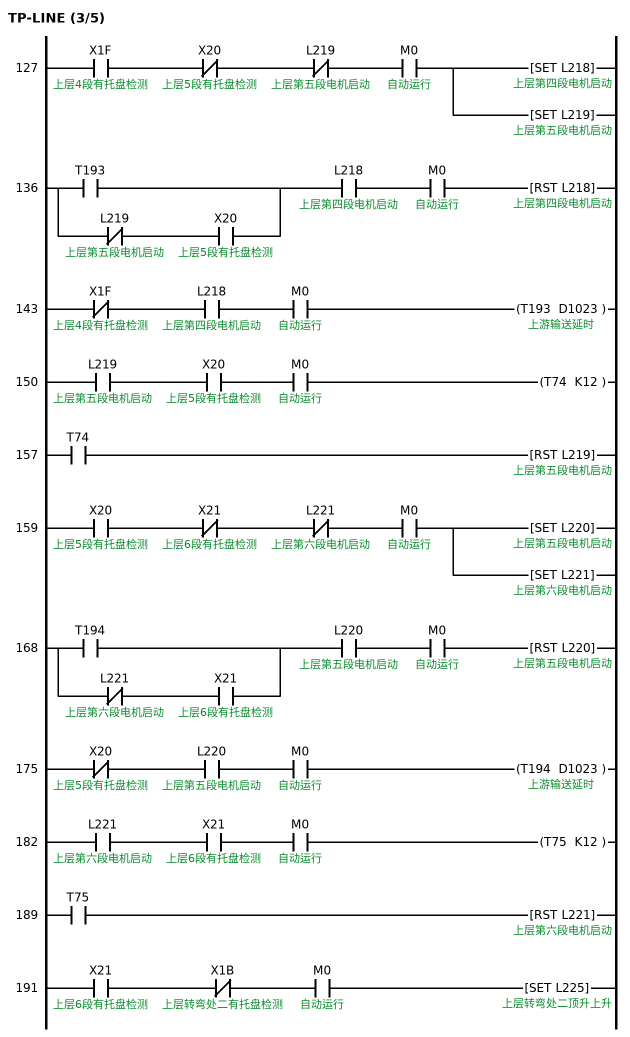
[picture p72: ladder of TP-LINE, rungs at steps 127 to 191]
127   LD      X1F  ; 上层4段有托盘检测
      ANI     X20  ; 上层5段有托盘检测
      ANI     L219  ; 上层第五段电机启动
      AND     M0  ; 自动运行
      SET     L218  ; 上层第四段电机启动
        [note] 5
      SET     L219  ; 上层第五段电机启动
136   LD      T193
      LDI     L219  ; 上层第五段电机启动
      AND     X20  ; 上层5段有托盘检测
      ORB
      AND     L218  ; 上层第四段电机启动
      AND     M0  ; 自动运行
      RST     L218  ; 上层第四段电机启动
143   LDI     X1F  ; 上层4段有托盘检测
      AND     L218  ; 上层第四段电机启动
      AND     M0  ; 自动运行
      OUT     T193 D1023  ; 上游输送延时
150   LD      L219  ; 上层第五段电机启动
      AND     X20  ; 上层5段有托盘检测
      AND     M0  ; 自动运行
      OUT     T74 K12
157   LD      T74
      RST     L219  ; 上层第五段电机启动
159   LD      X20  ; 上层5段有托盘检测
      ANI     X21  ; 上层6段有托盘检测
      ANI     L221  ; 上层第六段电机启动
      AND     M0  ; 自动运行
      SET     L220  ; 上层第五段电机启动
        [note] 6
      SET     L221  ; 上层第六段电机启动
168   LD      T194
      LDI     L221  ; 上层第六段电机启动
      AND     X21  ; 上层6段有托盘检测
      ORB
      AND     L220  ; 上层第五段电机启动
      AND     M0  ; 自动运行
      RST     L220  ; 上层第五段电机启动
175   LDI     X20  ; 上层5段有托盘检测
      AND     L220  ; 上层第五段电机启动
      AND     M0  ; 自动运行
      OUT     T194 D1023  ; 上游输送延时
182   LD      L221  ; 上层第六段电机启动
      AND     X21  ; 上层6段有托盘检测
      AND     M0  ; 自动运行
      OUT     T75 K12
189   LD      T75
      RST     L221  ; 上层第六段电机启动
191   LD      X21  ; 上层6段有托盘检测
      ANI     X1B  ; 上层转弯处二有托盘检测
      AND     M0  ; 自动运行
      SET     L225  ; 上层转弯处二顶升上升
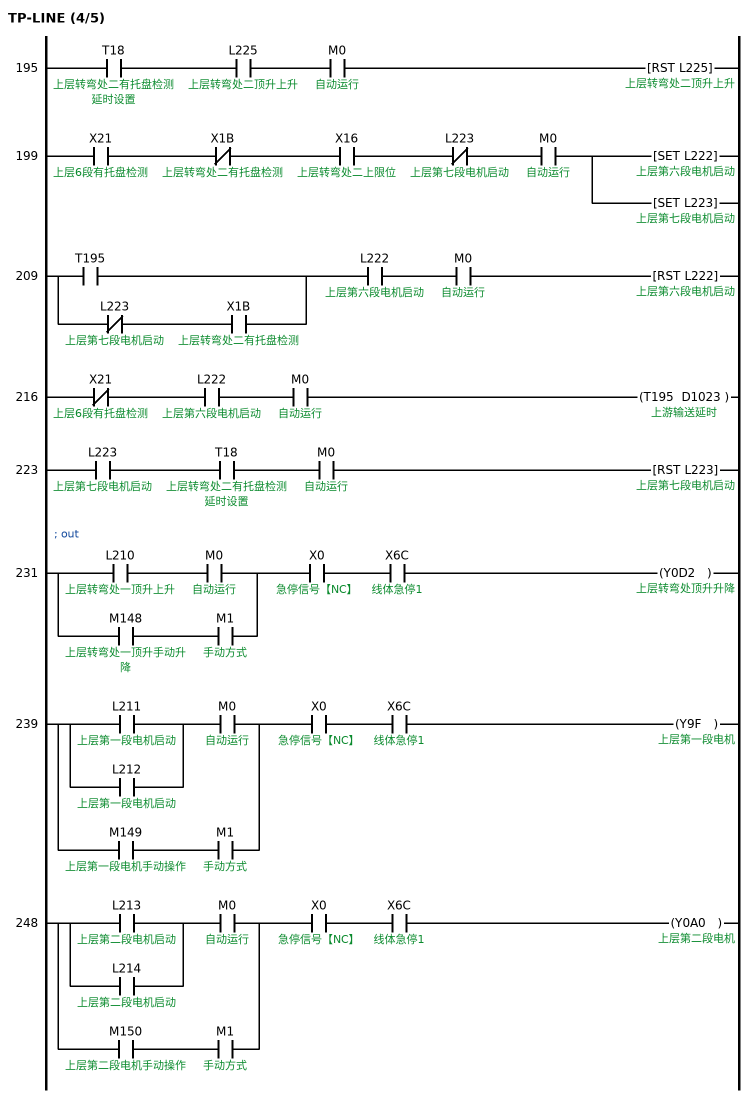
195   LD      T18  ; 上层转弯处二有托盘检测延时设置
      AND     L225  ; 上层转弯处二顶升上升
      AND     M0  ; 自动运行
      RST     L225  ; 上层转弯处二顶升上升
199   LD      X21  ; 上层6段有托盘检测
      ANI     X1B  ; 上层转弯处二有托盘检测
      AND     X16  ; 上层转弯处二上限位
      ANI     L223  ; 上层第七段电机启动
      AND     M0  ; 自动运行
      SET     L222  ; 上层第六段电机启动
        [note] 7
      SET     L223  ; 上层第七段电机启动
209   LD      T195
      LDI     L223  ; 上层第七段电机启动
      AND     X1B  ; 上层转弯处二有托盘检测
      ORB
      AND     L222  ; 上层第六段电机启动
      AND     M0  ; 自动运行
      RST     L222  ; 上层第六段电机启动
216   LDI     X21  ; 上层6段有托盘检测
      AND     L222  ; 上层第六段电机启动
      AND     M0  ; 自动运行
      OUT     T195 D1023  ; 上游输送延时
223   LD      L223  ; 上层第七段电机启动
      AND     T18  ; 上层转弯处二有托盘检测延时设置
      AND     M0  ; 自动运行
      RST     L223  ; 上层第七段电机启动
; out
231   LD      L210  ; 上层转弯处一顶升上升
      AND     M0  ; 自动运行
      LD      M148  ; 上层转弯处一顶升手动升降
      AND     M1  ; 手动方式
      ORB
      AND     X0  ; 急停信号【NC】
      AND     X6C  ; 线体急停1
      OUT     Y0D2  ; 上层转弯处顶升升降
239   LD      L211  ; 上层第一段电机启动
      OR      L212  ; 上层第一段电机启动
      AND     M0  ; 自动运行
      LD      M149  ; 上层第一段电机手动操作
      AND     M1  ; 手动方式
      ORB
      AND     X0  ; 急停信号【NC】
      AND     X6C  ; 线体急停1
      OUT     Y9F  ; 上层第一段电机
248   LD      L213  ; 上层第二段电机启动
      OR      L214  ; 上层第二段电机启动
      AND     M0  ; 自动运行
      LD      M150  ; 上层第二段电机手动操作
      AND     M1  ; 手动方式
      ORB
      AND     X0  ; 急停信号【NC】
      AND     X6C  ; 线体急停1
      OUT     Y0A0  ; 上层第二段电机
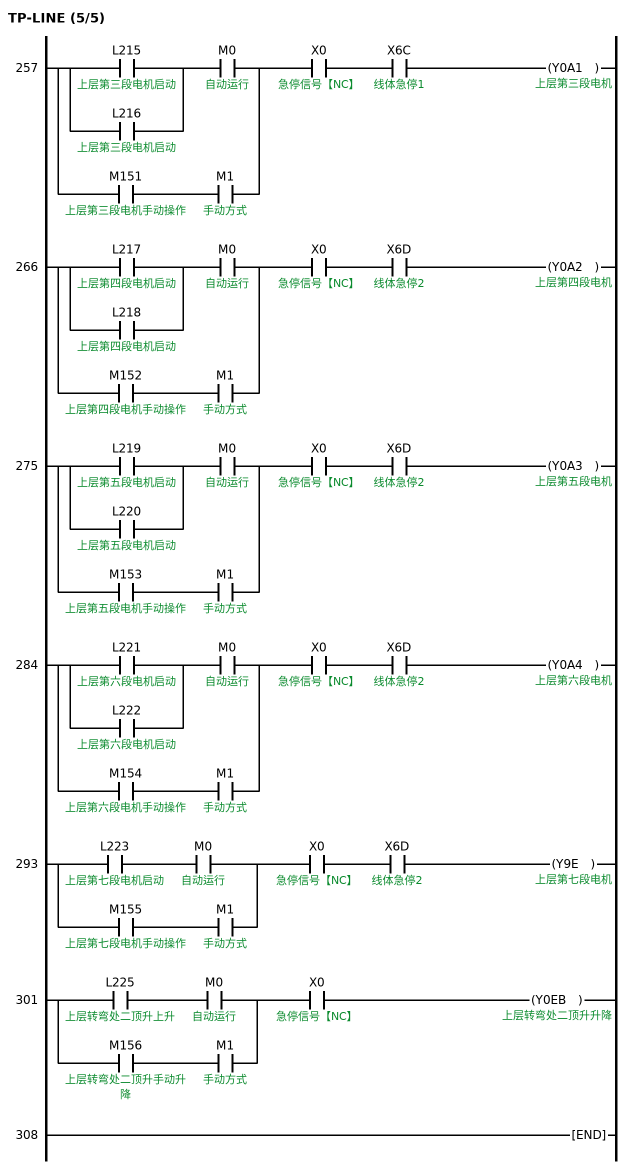
257   LD      L215  ; 上层第三段电机启动
      OR      L216  ; 上层第三段电机启动
      AND     M0  ; 自动运行
      LD      M151  ; 上层第三段电机手动操作
      AND     M1  ; 手动方式
      ORB
      AND     X0  ; 急停信号【NC】
      AND     X6C  ; 线体急停1
      OUT     Y0A1  ; 上层第三段电机
266   LD      L217  ; 上层第四段电机启动
      OR      L218  ; 上层第四段电机启动
      AND     M0  ; 自动运行
      LD      M152  ; 上层第四段电机手动操作
      AND     M1  ; 手动方式
      ORB
      AND     X0  ; 急停信号【NC】
      AND     X6D  ; 线体急停2
      OUT     Y0A2  ; 上层第四段电机
275   LD      L219  ; 上层第五段电机启动
      OR      L220  ; 上层第五段电机启动
      AND     M0  ; 自动运行
      LD      M153  ; 上层第五段电机手动操作
      AND     M1  ; 手动方式
      ORB
      AND     X0  ; 急停信号【NC】
      AND     X6D  ; 线体急停2
      OUT     Y0A3  ; 上层第五段电机
284   LD      L221  ; 上层第六段电机启动
      OR      L222  ; 上层第六段电机启动
      AND     M0  ; 自动运行
      LD      M154  ; 上层第六段电机手动操作
      AND     M1  ; 手动方式
      ORB
      AND     X0  ; 急停信号【NC】
      AND     X6D  ; 线体急停2
      OUT     Y0A4  ; 上层第六段电机
293   LD      L223  ; 上层第七段电机启动
      AND     M0  ; 自动运行
      LD      M155  ; 上层第七段电机手动操作
      AND     M1  ; 手动方式
      ORB
      AND     X0  ; 急停信号【NC】
      AND     X6D  ; 线体急停2
      OUT     Y9E  ; 上层第七段电机
301   LD      L225  ; 上层转弯处二顶升上升
      AND     M0  ; 自动运行
      LD      M156  ; 上层转弯处二顶升手动升降
      AND     M1  ; 手动方式
      ORB
      AND     X0  ; 急停信号【NC】
      OUT     Y0EB  ; 上层转弯处二顶升升降
308   END
END_PROGRAM

PROGRAM ServoScan
IF g_xScanStart  AND g_iXaxisNumber<>0 AND  g_iYaxisNumber<>0 THEN
	U10\G1500:=g_iXaxisNumber;
	U10\G1600:=g_iYaxisNumber;
	Y110:=NOT X114;
	Y111:=NOT X115;
END_IF;
END_PROGRAM

// device comments not shown above
X6  ; 急停1
X7  ; 急停2
X0B2  ; 上层开门信号
X0B3  ; 下层开门信号
X0B4  ; 下层出货完成信号
M52  ; 无原点提示
L60  ; 工位1-2送出输送速度
L140  ; 工位3-2送出输送速度
L224  ; 上层第七段电机启动
L226  ; 上层第三段电机启动
L227  ; 上层第二段电机启动
L252  ; 下层第十一段电机启动
T0  ; AB门上层出口段托盘到位无货延时
D436  ; 出口待机时间
D438  ; 上料待机时间
D456  ; 运行时间（分）
D522  ; 出口待机时间（分）
D534  ; 工作时间
D536  ; 故障率
D540  ; 稼动率
D544  ; 节拍
D550  ; 故障时间
D554  ; 运行-待机
D560  ; 工作时间
D564  ; 运行时间
D800  ; 延时时间设置
D801  ; 减速时间设定
D1051  ; AB门输送报警延时设置
